fbS2 ( bAutomat:=bAutomat, bManual:=bManual,bStop:=bStop,bReset:=bReset, bEnableMove:=bEnableMoveToS2,bBuffering:=bBuffering,
        bDriveMove:=fbS3.bDrivePrev, bSens1:=bSens1s02D2, bSens2:=bSens1s02D1,bSensFork:= bSens1s01D3, ConvStatusPrev1:=0,
        ConvStatusPrev2:=fbS1.ConvStatus, bButtConv:= bButt1s02, bButtConvRev:=bButt1s02Rev, bButtMove:=bButt1s01_s02,
         bDirect:=bDirect	,bReverse:=bReverse,   ConvStatusNext1:= fbS3.ConvStatus1, ConvStatusNext2:= fbS3.ConvStatus2,
		 bEnableMove3:=bEnableMove3_2(*fbDelayEnableMove3_2.Q*), bEnableMove2:= iCounterPallets>1,  //bSensFreePrev2:=fbS1.bSensFree,
	    bMove1:=bMove1s01_s02_1, bMove2:=bMove2, bMove3:=bMove1s02_1_s02_2, 
        bLongMove1=> bLongMove1s01_s02_1,bLongMove3=> bLongMove1s02_1_s02_2  );

	    bEnableMoveToS3:= NOT bMove1s03_2_s04_1 AND NOT bMove1s03_s04 AND NOT bMove1s01_s02_1 AND NOT bMove1s02_1_s02_2;
 
		
		bEnableMove3_3 := (fbS6.ConvStatus=0 OR fbS5.ConvStatus=0) AND fbS4.ConvStatus1=0 AND fbS4.ConvStatus2=0 
       AND NOT (bMove1s03_2_s04_1 OR bMove1s03_s04 OR bMove1s04_1_s04_2 OR bMove1s05_s06 OR bMove1s04_2_s05);
		  fbDelayEnableMove3_3(IN:=bEnableMove3_3, PT:=T#0.3S);
		  
fbS3 ( bAutomat:=bAutomat, bManual:=bManual,bStop:=bStop,bReset:=bReset, bEnableMove:=bEnableMoveToS3,bBuffering:=bBuffering,
        bDriveMove:=fbS4.bDrivePrev, bSens1:=bSens1s03D2, bSens2:=bSens1s03D1,ConvStatusPrev1:=fbS2.ConvStatus1,
        ConvStatusPrev2:=fbS2.ConvStatus2, bButtConv:= bButt1s03, bButtConvRev:=bButt1s03Rev, bButtMove:=bButt1s02_s03, 
		 bDirect:=bDirect	,bReverse:=bReverse,   ConvStatusNext1:= fbS4.ConvStatus1, ConvStatusNext2:= fbS4.ConvStatus2,
		 bEnableMove3:=fbDelayEnableMove3_3.Q,  bEnableMove2:= TRUE,  //bSensFreePrev1:=fbS2.bSensFree1, bSensFreePrev2:=fbS2.bSensFree2,
	    bMove1:=bMove1s02_2_s03_1, bMove2:=bMove1s02_s03, bMove3:=bMove1s03_1_s03_2, 
        bLongMove1=> bLongMove1s02_2_s03_1,bLongMove2=>bLongMove1s02_s03, bLongMove3=> bLongMove1s03_1_s03_2 );	  
	  
	    bEnableMoveToS4:= NOT bMove1s04_2_s05 AND NOT bMove1s02_2_s03_1 AND NOT bMove1s03_1_s03_2;
 
		
		
		bEnableMove3_4 := fbS6.ConvStatus=0 OR fbS5.ConvStatus=0 AND NOT (bMove1s05_s06 OR bMove1s04_2_s05);
		fbDelayEnableMove3_4(IN:=bEnableMove3_4, PT:=T#0.3S);
		
fbS4 ( bAutomat:=bAutomat, bManual:=bManual,bStop:=bStop,bReset:=bReset, bEnableMove:=bEnableMoveToS4,bBuffering:=bBuffering,
        bDriveMove:=fbS5.bDrivePrev AND bSens1s05D2, bSens1:=bSens1s04D2, bSens2:=bSens1s04D1,ConvStatusPrev1:=fbS3.ConvStatus1,
        ConvStatusPrev2:=fbS3.ConvStatus2, bButtConv:= bButt1s04, bButtConvRev:=bButt1s04Rev, bButtMove:=bButt1s03_s04,
         bDirect:=bDirect	,bReverse:=bReverse,   ConvStatusNext1:= fbS5.ConvStatus,
		 bEnableMove3:=fbDelayEnableMove3_4.Q,  bEnableMove2:= TRUE, // bSensFreePrev1:=fbS3.bSensFree1, bSensFreePrev2:=fbS3.bSensFree2,
	    bMove1:=bMove1s03_2_s04_1, bMove2:=bMove1s03_s04, bMove3:=bMove1s04_1_s04_2, 
         bLongMove1=>bLongMove1s03_2_s04_1,bLongMove2=>bLongMove1s03_s04, bLongMove3=> bLongMove1s04_1_s04_2  );	  
	
  		
		bEnableRead := NOT bMove1s05_s06 AND NOT bMove1s03_2_s04_1 AND NOT bMove1s04_1_s04_2 AND NOT bMove1s03_s04 ;
		
fbLoadScan (bAutomat:=bAutomat,bEnable:=bEnableRead, iConvStatus:=fbS4.ConvStatus2, 
        sInID:=sScanID_1, stLoad:=stLoadS4_1, bReadScan:=bReadScan_1, 
        bRequestID=>bRequestID_1,bEnableReadyID=>bEnableReadyID, bOverflowID=>bOverflow_CTU_ID1,
		bSetVal:=bSetVal_ID1, bResetCTU:=bResetCTU_ID1, bCountNoRead=>bCountNoRead_ID1);		 
		
						
	    bEnableMoveToS5:= NOT bMove1s05_s06 AND NOT bMove1s03_2_s04_1 AND NOT bMove1s04_1_s04_2  AND bEnableReadyID;
	  
fbS5 ( bAutomat:=bAutomat, bManual:=bManual,bStop:=bStop,bReset:=bReset, bEnableMove:= bEnableMoveToS5,
        bDriveMove:=fbS6.bDrivePrev, bSens1:=bSens1s05D2, bSens2:=bSens1s05D1, bStopSecPlace:=TRUE,
        bButtConv:= bButt1s05,bButtConvRev:=bButt1s05Rev, ConvStatusPrev := fbS4.ConvStatus2,
		 bDirect:=bDirect	,bReverse:=bReverse,
		bSensFreePrev:= bSens1s04D1, bMove:=bMove1s04_2_s05,bLongMove=>bLongMove1s04_2_s05, );  
	  	
	
		bEnableWeight := NOT bMove1s04_2_s05 AND NOT bMove1s05_s06 ;
		
fbLoadWeight (bAutomat:=bAutomat,bEnable:=bEnableWeight,bMove:=bMove1s04_2_s05, iConvStatus:=fbS5.ConvStatus, stLoadIn:=stLoadS4_1,
        (*sInWeight:=sWeight_1*)rInWeight:= Massa_1_Gramms   ,  stLoad:=stLoadS5_1, stLoadMove:=stLoadS4_5_1, 
        (*bRequestWeight=>bRequestWeight_1,*) bEnableReadyData=>bEnableReadyData, bOverflowWeight=>bOverflow_CTU_Weight1,
		  bCountNoReadWeight=>bCountNoRead_Weight1, bSetValWeight:=bSetVal_Weight1, bResetCTUWeight:=bResetCTU_Weight1);	
		
			
	    bEnableMoveToS6:= NOT bMove1s04_2_s05   AND bEnableReadyData ;
	  
fbS6 ( bAutomat:=bAutomat, bManual:=bManual,bStop:=bStop,bReset:=bReset, bEnableMove:= bEnableMoveToS6,
        bSens1:=TRUE, bSens2:=bSens1s06D1, (*bSensFork:= bSens1s06D2, *)bButtConv:= bButt1s06, bButtConvRev:=bButt1s06Rev,
		 bDirect:=bDirect	,bReverse:=bReverse,bLastPlace:=TRUE,bLongMove=>bLongMove1s05_1s06,
	    bMove:=bMove1s05_s06,ConvStatusPrev := fbS5.ConvStatus,bSensFreePrev := bSensFreePrevS6);  
		
		bSensFreePrevS6 := fbS6.ConvStatus = 0;
		
		
fbLoadDataToWMS(bAutomat:=bAutomat,stLoadIn:=stLoadS5_1, bEnable:=NOT bMove1s05_s06, 
iConvStatus:=fbS6.ConvStatus, bMove	:=bMove1s05_s06, stLoadMove:=  stLoadS5_6_1, stLoad:=stLoadS6_1,
sMessageOut=>sMessageOut1, bMessageReady:=bMessageReady1	);		
		
		
	  
bDrive1s01M1    := fbS1.bDrive 		AND bDirect ;
bDrive1s01M1Rev := fbS1.bDriveRev 		AND bReverse AND bSens1s01D2;
bDrive1s02M1    := fbS2.bDrive 		AND bDirect ;
bDrive1s02M1Rev := fbS2.bDriveReverse 	AND bReverse;
bDrive1s03M1    := fbS3.bDrive 		AND bDirect ;
bDrive1s03M1Rev := fbS3.bDriveReverse 	AND bReverse;
bDrive1s04M1    := fbS4.bDrive 		AND bDirect ;
bDrive1s04M1Rev := fbS4.bDriveReverse 	AND bReverse;  
bDrive1s05M1    := fbS5.bDrive 		AND bDirect ;
bDrive1s05M1Rev := fbS5.bDriveRev 		AND bReverse;
bDrive1s06M1    := fbS6.bDrive 		AND bDirect AND bSens1s06D1;
bDrive1s06M1Rev := fbS6.bDriveRev 		AND bReverse;

END_PROGRAM

// ---- POUs/FB/FBconv/FB_ConvPlace.TcPOU
FUNCTION_BLOCK FB_ConvPlace
VAR_INPUT
	bFirstPlace:BOOL:=FALSE;
	bLastPlace:BOOL:=FALSE;
	bAutomat: BOOL;
	bStopSecPlace: BOOL;
	bEnableMove: BOOL;
	ConvStatusPrev: BYTE;
	bManual: BOOL;
	bDriveMove: BOOL;
	bSens1: BOOL;
	bSens2: BOOL;
	bSens3: BOOL := TRUE;
	bSensFork: BOOL := FALSE;
	tBusy: TIME := TIME#10ms;
	tFree: TIME := TIME#2s800ms;
	tLongMove: TIME := TIME#15s0ms;
	bReset: BOOL := FALSE;
	bStop: BOOL;
	bSensFreePrev: BOOL;
	bSensFreeNext: BOOL;
	bButtConv: BOOL;
	bButtConvRev: BOOL;
	bButtMove: BOOL;
	 bDirect: BOOL;
	bReverse: BOOL;
END_VAR
VAR_OUTPUT
	bDrive: BOOL;
	bDriveRev: BOOL;
	ConvStatus: BYTE;
	bDrivePrev: BOOL;
	bLongMove: BOOL;
	bSensFree: BOOL;
	bReqMove: BOOL;
	bForkFree: BOOL;
END_VAR
VAR
	fbBusy1: FB_Busy1;
	fbBusy2: FB_Busy1;
	fbBusy3: FB_Busy1;
	fbBusyFork: FB_Busy2;
	fbButt: FB_ButtonToggle;
	fbButtRev: FB_ButtonToggle;
	bDriveManu: BOOL;
	bResManu: BOOL;
	bDriveManuRev: BOOL;
	fbLongMove: TON;
	bDriveConv: BOOL;
	fbButtMove: R_TRIG;
	bDriveConvRev: BOOL;
END_VAR
VAR_IN_OUT
	bMove: BOOL;
END_VAR






     (* определение заполненности конвейерного места*)
    fbBusy1 ( bSens:= bSens1,  tFree:=  tFree ,   tBusy:= tBusy , Reset := bReset ) ;
	fbBusy2 ( bSens:= bSens2,  tFree:=   tFree ,   tBusy:=  tBusy , Reset := bReset ) ;
	fbBusy3 ( bSens:= bSens3,  tFree:=   tFree ,   tBusy:=  tBusy , Reset := bReset ) ;
	fbBusyFork( bSens:= bSensFork,  tFree:=   T#10s ,   tBusy:= T#0s , Reset := bReset ) ;
	IF  NOT fbBusy1.ConvBusy AND NOT  fbBusy2.ConvBusy AND NOT  fbBusy3.ConvBusy THEN ConvStatus := 0;
	ELSIF fbBusy1.ConvBusy AND NOT  fbBusy2.ConvBusy THEN ConvStatus := 1;
	ELSIF NOT  fbBusy1.ConvBusy AND   fbBusy2.ConvBusy THEN ConvStatus := 2;
	ELSIF fbBusy1.ConvBusy AND   fbBusy2.ConvBusy THEN ConvStatus := 3;
	END_IF
	
	bForkFree:= NOT fbBusyFork.ConvBusy;
	
	bSensFree:= bSens1 AND bSens2 AND bSens3;
	
	(* включение двигателя*)
     bDrive:= NOT bStop AND (  bDriveMove OR bDriveConv  OR  bDriveManu );
	  bDriveRev:= NOT bStop AND bDriveManuRev;
	
    (* включение двигателя в ручном режиме *)
	bResManu := bReset OR NOT bManual ;
	fbButt (bButt := bButtConv , bEnable := bManual AND NOT bDriveManuRev AND bDirect , bReset := bResManu OR NOT bDirect
OR bDirect AND bLastPlace AND NOT bSens2)  ;
     bDriveManu := fbButt.bOutB;
	fbButtRev (bButt := bButtConvRev  , bEnable :=  bManual  AND NOT bDriveManu AND bReverse, bReset := bResManu OR NOT bReverse
OR bReverse AND bFirstPlace AND NOT bSens1)  ;
 bDriveManuRev := fbButtRev.bOutB;

	(* включение перемещения*)

bReqMove:= bAutomat  AND  (ConvStatusPrev = 2  OR ConvStatusPrev =3) AND ConvStatus =0 AND  NOT fbBusyFork.ConvBusy ;

	IF    bEnableMove   AND  bReqMove
	 THEN  bMove := TRUE ;
	END_IF
	
	(* включение двигателей при перемещении *)
	bDriveConv:=   NOT bStop AND bMove  AND NOT  (ConvStatus = 2 OR ConvStatus = 3)  ;
	bDrivePrev := NOT bStop AND bMove AND NOT  (ConvStatus = 2 OR ConvStatus = 3) AND NOT (ConvStatusPrev = 0) ;
	

	
	
	(* выключение перемещения*)
	IF   bMove  AND ((*ConvStatusPrev = 0*) bSensFreePrev  OR bStopSecPlace ) AND  (ConvStatus = 2 OR ConvStatus = 3)  THEN bMove := FALSE ;
	END_IF
	
	(* долгое перемещение*)
	fbLongMove(IN := NOT bStop AND bMove , PT := tLongMove);
	 bLongMove:= fbLongMove.Q;
	 
	 (* включение-выключение перемещения кнопкой*)
	 
	fbButtMove (CLK :=bButtMove (*AND bManual*));
	IF fbButtMove.Q AND bManual THEN IF   NOT bMove  THEN bMove := TRUE;
         ELSIF bMove THEN  
      bMove := FALSE;
	END_IF
    END_IF
		
		


	 
		
		
	 IF bReset THEN 
     bMove := FALSE ; 
	  END_IF

END_FUNCTION_BLOCK

// ---- POUs/FB/FBauxiliary/FB_Busy1.TcPOU
FUNCTION_BLOCK FB_Busy1
VAR_INPUT
	bSens	 :BOOL;
	tBusy	 :TIME;
	tFree	 :TIME;
	Reset	 :BOOL;
END_VAR
VAR_OUTPUT
	ConvBusy :BOOL := TRUE;
END_VAR
VAR
	Timer1	 :TON;
	Timer2	 :TON;
END_VAR

Timer1 (IN := NOT bSens, PT := tBusy);
IF Timer1.Q THEN ConvBusy := TRUE;
END_IF
Timer2 (IN :=     bSens, PT := tFree);
IF Timer2.Q (*OR Reset*) THEN ConvBusy := FALSE;
END_IF

END_FUNCTION_BLOCK

// ---- POUs/FB/FBauxiliary/FB_Busy2.TcPOU
FUNCTION_BLOCK FB_Busy2
VAR_INPUT
	bSens	 :BOOL;
	tBusy	 :TIME;
	tFree	 :TIME;
	Reset	 :BOOL;
END_VAR
VAR_OUTPUT
	ConvBusy :BOOL;
END_VAR
VAR
	Timer1	 :TON;
	Timer2	 :TON;
END_VAR

Timer1 (IN := 	  bSens, PT := tBusy);
IF Timer1.Q THEN ConvBusy := TRUE;
END_IF
Timer2 (IN := NOT bSens, PT := tFree);
IF Timer2.Q (*OR Reset*) THEN ConvBusy := FALSE;
END_IF

END_FUNCTION_BLOCK

// ---- POUs/FB/FBconv/FB_ConvPlaceDouble.TcPOU
FUNCTION_BLOCK FB_ConvPlaceDouble
VAR_INPUT
	bStopSecPlace: BOOL;
	bStartAutomat: BOOL;
	bAutomat: BOOL;
	bManual: BOOL;
	bReset: BOOL := FALSE;
	bStop: BOOL;
	bEnableMove: BOOL;
	ConvStatusPrev1: BYTE;
	ConvStatusPrev2: BYTE;
	bDriveMove: BOOL;
	bButtConv: BOOL;
	bButtConvRev: BOOL;
	bButtMove: BOOL;
	bSens1: BOOL;
	bSens2: BOOL;
	bSens3: BOOL := TRUE;
	bSensFork: BOOL := FALSE;
	tBusy: TIME := TIME#10ms;
	tFree: TIME := TIME#2s800ms;
	tLongMove: TIME := TIME#30s0ms;
	bBuffering: BOOL;
	 bDirect: BOOL;
	bReverse: BOOL;
	ConvStatusNext1: BYTE;
	ConvStatusNext2: BYTE;
	bEnableMove3:BOOL;
	bEnableMove2:BOOL;
	
	bSensFreePrev1:BOOL;
	bSensFreePrev2:BOOL;
END_VAR
VAR_OUTPUT
	bDrive: BOOL;
	bDriveReverse: BOOL;
	ConvStatus2: BYTE;
	ConvStatus1: BYTE;
	bDrivePrev: BOOL;
	bLongMove1: BOOL;
	bLongMove2: BOOL;
	bLongMove3: BOOL;
	bSensFree1:BOOL;
	bSensFree2:BOOL;
END_VAR
VAR
	fbBusy1: FB_Busy1;
	fbBusy2: FB_Busy1;
	fbBusyFork: FB_Busy2;
	fbButt: FB_ButtonToggle;
	fbButtReverse: FB_ButtonToggle;
	bDriveManu: BOOL;
	bResManu: BOOL;
	bDriveManuReverse: BOOL;
	bDriveConv1: BOOL;
	bDriveConv2: BOOL;
	bDriveConv3: BOOL;
	bDriveConv: BOOL;
	bDrivePrev1: BOOL;
	bDrivePrev2: BOOL;
	fbLongMove1: TON;
	fbLongMove2: TON;
	fbLongMove3: TON;
	fbButtMove: R_TRIG;
	fbStartAutomat: R_TRIG;
	bStartConv: BOOL;
	fbConvBusy1Puls: R_TRIG;
	fbConvBusy2Puls: R_TRIG;
	fbStartTimer: TON;
	fbFinStartAutomat: F_TRIG;
	bPermMove1: BOOL;
	bPermMove2: BOOL;
	bPermMove3: BOOL;

END_VAR
VAR_IN_OUT
	bMove1: BOOL;
	bMove2: BOOL;
	bMove3: BOOL;
END_VAR

fbBusy1 ( bSens := bSens1, tFree := tFree, tBusy := tBusy, Reset := bReset);
fbBusy2 ( bSens := bSens2, tFree := tFree, tBusy := tBusy, Reset := bReset);
fbBusyFork( bSens:= bSensFork,  tFree:=   T#10S ,   tBusy:= T#0S , Reset := bReset ) ;

 bSensFree1:= bSens1;    
 bSensFree2:= bSens2; 

IF NOT fbBusy1.ConvBusy THEN ConvStatus1 := 0;
	ELSE
		ConvStatus1 := 2;
END_IF

IF NOT fbBusy2.ConvBusy  THEN ConvStatus2 := 0;
	ELSE
		ConvStatus2 := 2;
END_IF

bDrive := NOT bStop AND (bDriveMove OR bDriveConv OR bDriveManu OR bStartConv);
bDriveReverse := NOT bStop AND bDriveManuReverse;

bResManu := bReset OR NOT bManual;
fbButt (bButt := bButtConv AND bManual AND NOT bDriveManuReverse AND bDirect, bReset := bResManu  OR NOT bDirect); 
bDriveManu := fbButt.bOutB;
fbButtReverse (bButt := bButtConvRev AND bManual AND NOT bDriveManu AND bReverse, bReset := bResManu  OR NOT bReverse);
 bDriveManuReverse := fbButtReverse.bOutB;

(* Перемещения*)
(* Условия включения перемещения*)
bPermMove1:= ConvStatusPrev1=0 AND ConvStatus2=0  AND NOT bMove2  AND NOT bMove3;

IF  bAutomat AND bEnableMove AND bPermMove1 AND (ConvStatusPrev2 = 2 OR ConvStatusPrev2 = 3) AND ConvStatus1 = 0 AND  NOT fbBusyFork.ConvBusy
	THEN  bMove1 := TRUE;
END_IF

(* Выключение перемещения bMove1*)
IF  bMove1 AND (ConvStatusPrev2 = 0 OR bStopSecPlace (*OR bSensFreePrev2*)) AND (ConvStatus1 = 2 OR ConvStatus1 = 3) THEN bMove1 := FALSE;
END_IF





bPermMove2 := (( ConvStatusPrev1=2 OR ConvStatusPrev1=3) AND ConvStatus1=0 OR  ConvStatusPrev1=0 AND  (ConvStatus1 = 2 OR
ConvStatus1 = 3)) AND NOT bMove1  AND NOT bMove3 AND bEnableMove2;

IF  bAutomat AND bEnableMove AND bPermMove2 AND (ConvStatusPrev2 = 2 OR ConvStatusPrev2 = 3) AND ConvStatus2 = 0 
	THEN  bMove2 := TRUE;
END_IF


(* Выключение перемещения bMove2*)
IF  bMove2 AND (ConvStatusPrev2 = 0 OR bStopSecPlace (*OR bSensFreePrev2*)) AND (ConvStatus2 = 2 OR ConvStatus2 = 3) THEN bMove2 := FALSE;
END_IF

//bPermMove3 := (ConvStatusNext1=0 AND ConvStatusNext2=0  OR (ConvStatusNext1=2 OR ConvStatusNext1=3) AND ConvStatusNext2=0 )
//AND NOT bMove1 AND NOT bMove2;
bPermMove3 := (NOT (( ConvStatusPrev2=2 OR ConvStatusPrev2=3) AND ConvStatusPrev1=0) AND NOT bBuffering OR
bBuffering AND 	bEnableMove3)  AND NOT bMove1 AND NOT bMove2;

IF  bAutomat AND bEnableMove AND bPermMove3 AND (ConvStatus1 = 2 OR ConvStatus1 = 3) AND ConvStatus2 = 0 
	THEN bMove3 := TRUE;
END_IF

(* Выключение перемещения bMove3*)
IF  bMove3 AND (ConvStatus1 = 0 OR bStopSecPlace (*OR bSens1*)) AND (ConvStatus2 = 2 OR ConvStatus2 = 3) THEN bMove3 := FALSE;
END_IF




(* Включение двигателей *)
bDriveConv1 := NOT bStop AND bMove1 AND NOT (ConvStatus1 = 2 OR ConvStatus1 = 3);
bDriveConv2 := NOT bStop AND bMove2 AND NOT (ConvStatus2 = 2 OR ConvStatus2 = 3);
bDriveConv3 := NOT bStop AND bMove3 AND NOT (ConvStatus2 = 2 OR ConvStatus2 = 3);
	
bDriveConv := bDriveConv1 OR bDriveConv2 OR bDriveConv3;

bDrivePrev1 := NOT bStop AND bMove1 AND NOT (ConvStatus1 = 2 OR ConvStatus1 = 3) AND NOT (ConvStatusPrev2 = 0);
bDrivePrev2 := NOT bStop AND bMove2 AND NOT (ConvStatus2 = 2 OR ConvStatus2 = 3) AND NOT ((ConvStatusPrev1 = 0)AND(ConvStatusPrev2 = 0)) ;
	
bDrivePrev := bDrivePrev1 OR bDrivePrev2 ;

(* Долгое перемещение*)
fbLongMove1(IN := NOT bStop AND bMove1, PT := tLongMove);
bLongMove1 := fbLongMove1.Q;
fbLongMove2(IN := NOT bStop AND bMove2, PT := tLongMove);
bLongMove2 := fbLongMove2.Q;
fbLongMove3(IN := NOT bStop AND bMove3, PT := tLongMove);
bLongMove3 := fbLongMove3.Q;

(* Включение-выключение перемещения кнопкой*)
fbButtMove (CLK :=bButtMove (*AND bManual*));
IF fbButtMove.Q THEN 
	IF NOT bMove2 AND bManual THEN bMove2 := TRUE;
		ELSIF bMove2 THEN  
      bMove2 := FALSE;
	END_IF
   // bButtMove := FALSE;
END_IF

IF  bReset THEN bMove1 := FALSE; bMove2 := FALSE; bMove3 := FALSE; bStartConv := FALSE; 
	
END_IF

(*
(* Начальный режим*)
	fbStartAutomat (CLK := bStartAutomat);
IF 	fbStartAutomat.Q THEN 
IF NOT bReverse 
THEN 
IF (ConvStatus1=2 OR ConvStatus1=3)AND ConvStatusNext =1          THEN
	bStartConvReverse := TRUE;
END_IF

ELSE  bStartConvReverse := TRUE;
(* IF  NOT (ConvStatus1=2 OR ConvStatus1=3)AND ConvStatusNext =1 
THEN  bStartConvReverse := TRUE;
END_IF*)
END_IF
END_IF

	fbConvBusy1Puls (CLK := fbBusy1.ConvBusy);
//	fbConvBusy2Puls (CLK := fbBusy2.ConvBusy);

//	fbStartTimer (IN := bStartConv, PT := tStartTimer);
	fbStartTimerReverse (IN := bStartConvReverse, PT := tStartTimer);

(*IF    (bFinalConv  AND (ConvStatus = 3 OR ConvStatus = 2) OR NOT bFinalConv AND ((ConvStatus = 3 OR ConvStatus = 2) AND (ConvStatusNext = 3 OR ConvStatusNext = 2)) OR fbConvBusy2Puls.Q OR fbStartTimer.Q)
OR NOT bStartAutomat THEN  bStartConv := FALSE;
END_IF*)

IF 	  (bStartConvReverse AND (bFinalConvReverse AND (ConvStatus = 3 OR ConvStatus = 1) OR NOT bFinalConvReverse AND ((ConvStatus = 3 OR ConvStatus = 1) AND (ConvStatusPrev = 3 OR ConvStatusPrev = 1)) OR fbConvBusy1Puls.Q OR fbStartTimerReverse.Q))
OR NOT bStartAutomat THEN bStartConvReverse := FALSE;
END_IF

fbFinStartAutomat(CLK:=bStartAutomat);
IF fbFinStartAutomat.Q AND (ConvStatus1=2 OR ConvStatus1=3)AND ConvStatusNext =1   THEN
	bMoveReverse:=TRUE;
END_IF
*)

END_FUNCTION_BLOCK

// ---- POUs/ProcessingLoadData/FB_LoadScan.TcPOU
FUNCTION_BLOCK FB_LoadScan
VAR_INPUT
	bEnable			:BOOL;
	iConvStatus		:BYTE;
	bAutomat		:BOOL;
	
	bResetCTU		:BOOL;		
	bSetVal			:WORD;			
END_VAR
VAR_OUTPUT
	bEnableReadyID	:BOOL;
	bRequestID		:BOOL;
	bCountNoRead	:WORD;		//Кол-во несчитываний
	bOverflowID		:BOOL;		//Переполнение счетчика несчитываний ID
END_VAR
VAR
	fbPulsRequest	:R_TRIG;
	bStartRequest	:BOOL;
	fbDelayRead		:TON;
	WaitingID		:TON;
	bNoRead			:BOOL;		//Несчитывание
	bWriteIDgood	:BOOL;
	fbPulsNoread 	:R_TRIG;
	CTU 			:CTU;		//Счетчик
END_VAR
VAR_IN_OUT	
	stLoad			:ST_LoadData;
	bReadScan		:BOOL;
	sInID			:STRING;
END_VAR


bStartRequest:= bEnable AND bAutomat AND (iConvStatus=2 OR iConvStatus=3);

bEnableReadyID 	R= NOT bStartRequest;
bRequestID 	   	R= NOT bStartRequest  OR bReadScan;
bNoRead 		R= NOT bStartRequest;
bWriteIDgood    R= NOT bStartRequest;

fbPulsRequest(CLK:=bStartRequest);
IF fbPulsRequest.Q THEN
	bRequestID:=TRUE;
	bReadScan:=FALSE;
END_IF

fbDelayRead(IN:=bReadScan, PT:=T#0.3S);

WaitingID(IN:= bRequestID , PT:=T#3S);
bNoRead S= WaitingID.Q ;

fbPulsNoread(CLK:=bNoRead);

CTU(CU:=fbPulsNoread.Q, RESET:=bResetCTU, PV:=bSetVal);
bCountNoRead:=CTU.CV;

IF bReadScan AND NOT (bCountNoRead>=bSetVal) THEN
	stLoad.sID:= sInID;
	
	IF stLoad.sID<>'' OR fbDelayRead.Q THEN	
		bWriteIDgood:=TRUE;
		bReadScan:=FALSE;
	END_IF	
END_IF
bEnableReadyID S= bWriteIDgood OR bNoRead;

IF iConvStatus=0 THEN
	stLoad.sID:= '';
	stLoad.sWeight:= '';
	sInID:='';
END_IF

(*IF bCountNoRead>=bSetVal THEN bOverflowID:=TRUE;
	ELSE bOverflowID:=FALSE;
END_IF*)

END_FUNCTION_BLOCK

// ---- POUs/ProcessingLoadData/FB_LoadWeight.TcPOU
FUNCTION_BLOCK FB_LoadWeight
VAR_INPUT
	stLoadIn			:ST_LoadData;
	bEnable				:BOOL;
	iConvStatus			:BYTE;
	bAutomat			:BOOL;
	
	rInWeight			:DINT;;
	bMove				:BOOL;
	bReadWeight     	:BOOL;
	
	bResetCTUWeight		:BOOL;	//Очистка счетчика невзвешиваний	
	bSetValWeight		:WORD;	//Заданное значение разрешенных ошибок
END_VAR
VAR_OUTPUT
	bEnableReadyData	:BOOL;
	bRequestWeight		:BOOL;
	bCountNoReadWeight	:WORD;		//Кол-во несчитываний
	bOverflowWeight		:BOOL;		//Переполнение счетчика несчитываний весов
END_VAR
VAR
	fbPulsRequest		:R_TRIG;
	bStartRequest		:BOOL;
	fbPulsReadWeight	:R_TRIG;
	fbDelayWeight		:TON;
	fbStartMove			:R_TRIG;
	fbFinMove			:F_TRIG;
	bReadySt			:BOOL;
	bStartMove			:BOOL;
	bEndMove			:BOOL;
	sInWeight			:STRING;
	
	WaitingWeight		:TON;
	bNoReadWeight		:BOOL;		//Несчитывание
	bWriteWeightGood	:BOOL;
	fbPulsNoreadWeight 	:R_TRIG;
	CTU 				:CTU;		//Счетчик
END_VAR

VAR_IN_OUT
	stLoadMove      	:ST_LoadData;
	stLoad				:ST_LoadData;
//	bReadWeight			:BOOL;
END_VAR

fbStartMove(CLK:=bMove);
bStartMove S=fbStartMove.Q;
IF bStartMove THEN 
	stLoadMove := stLoadIn;
	IF stLoadMove.sID=stLoadIn.sID  AND stLoadMove.sWeight=stLoadIn.sWeight  THEN
		bStartMove:=FALSE;
	END_IF
END_IF

fbFinMove(CLK:=bMove);
bEndMove S= fbFinMove.Q;
IF bEndMove THEN 
	stLoad := stLoadMove;
	IF stLoadMove.sID=stLoad.sID  AND stLoadMove.sWeight=stLoad.sWeight  THEN
		bEndMove:=FALSE;
	END_IF
END_IF
//bReadySt := stLoad.sID = stLoadIn.sID  AND stLoad.sWeight = stLoadIn.sWeight;

bStartRequest:= bEnable AND bAutomat AND (iConvStatus=2 OR iConvStatus=3) AND NOT bEndMove;

bEnableReadyData 	R= NOT bStartRequest;
bRequestWeight 		R= NOT bStartRequest;
bNoReadWeight		R= NOT bStartRequest;

fbPulsRequest(CLK:=bStartRequest);
IF fbPulsRequest.Q THEN
	bRequestWeight:=TRUE;
END_IF

WaitingWeight(IN:= bRequestWeight, PT:=T#2S);
bNoReadWeight S= WaitingWeight.Q ;

fbPulsNoreadWeight(CLK:=bNoReadWeight);

CTU(CU:=fbPulsNoreadWeight.Q, RESET:=bResetCTUWeight, PV:=bSetValWeight);
bCountNoReadWeight:=CTU.CV;

fbDelayWeight(IN:=bRequestWeight(*bReadWeight*), PT:=T#0.3S);

sInWeight:= DINT_TO_STRING(rInWeight);
IF bRequestWeight(*bReadWeight  AND bReadySt*)AND NOT (bCountNoReadWeight=bSetValWeight) THEN
	stLoad.sWeight:= sInWeight;
	
	IF stLoad.sWeight<>'' OR fbDelayWeight.Q THEN	
		bWriteWeightGood	:=TRUE;	
		bRequestWeight		:=FALSE;
	END_IF	
END_IF

bEnableReadyData S= bWriteWeightGood OR bNoReadWeight;

IF iConvStatus=0 THEN
	stLoad.sID:= '';
	stLoad.sWeight:= '';
END_IF

IF bCountNoReadWeight>=bSetValWeight THEN bOverflowWeight:=TRUE;
	ELSE bOverflowWeight:=FALSE;
END_IF

END_FUNCTION_BLOCK

// ---- POUs/ExchangeWMS/FB_LoadDataToWMS.TcPOU
FUNCTION_BLOCK FB_LoadDataToWMS
VAR_INPUT
	stLoadIn		:ST_LoadData;
	bEnable			:BOOL;
	iConvStatus		:BYTE;
	bAutomat		:BOOL;
	bMove			:BOOL;
	
END_VAR
VAR_OUTPUT
	sMessageOut:T_MaxString;
	
END_VAR
VAR
	fbStartMove		:R_TRIG;
	fbFinMove		:F_TRIG;
	
	bStartMove:BOOL;
	bEndMove:BOOL;
	fbDelayStartMove:TON;
	fbDelayFinMove:TON;
	bReadySend: BOOL;
	
	fbCreateMessage: FB_CreateMessage;
END_VAR
VAR_IN_OUT
	stLoadMove      :ST_LoadData;
	stLoad			:ST_LoadData;
     bMessageReady:BOOL;
END_VAR

fbStartMove(CLK:=bMove);
bStartMove S=fbStartMove.Q;
fbDelayStartMove(IN:=bStartMove,PT:=T#0.3S);
IF bStartMove THEN 
	stLoadMove := stLoadIn;
	IF stLoadMove.sID=stLoadIn.sID  AND  stLoadMove.sWeight=stLoadIn.sWeight OR fbDelayStartMove.Q  THEN
		bStartMove:= FALSE;
	END_IF
END_IF


fbFinMove(CLK:=bMove);
bEndMove S= fbFinMove.Q;
fbDelayFinMove(IN:=bEndMove,PT:=T#0.3S);
IF bEndMove THEN 
	stLoad := stLoadMove;
	IF stLoadMove.sID=stLoad.sID   AND  stLoadMove.sWeight=stLoad.sWeight  OR fbDelayFinMove.Q  THEN
		bEndMove:= FALSE;
	END_IF
END_IF


bReadySend:=bAutomat AND (iConvStatus=2 OR iConvStatus=3) AND NOT bEndMove;

fbCreateMessage(stLoad:=stLoad, bCreateMessage:=bReadySend, sMessageOut=>sMessageOut,
bMessageReady:= bMessageReady );

END_FUNCTION_BLOCK

// ---- POUs/ExchangeWMS/FB_CreateMessage.TcPOU
FUNCTION_BLOCK FB_CreateMessage
VAR_INPUT
	stLoad		:ST_LoadData;
	bCreateMessage :BOOL;
END_VAR
VAR_OUTPUT
	sMessageOut:T_MaxString;
	
END_VAR
VAR
sTemplateMessage:T_MaxString:='|MsgNam=WMS.TEGEW|TrxId=|RFIDNAM=|DzTrn=|ArtGewBru=|';
fbPulsCreateMessage:R_TRIG;
sTrxId:STRING;
i :INT;
sMessage :T_MaxString;
iPosRFID:INT;
iPosTime:INT;
iPosBrutto:INT;
	

fbFileOpen:FB_FileOpen;
END_VAR
VAR PERSISTENT
iCountTrxId: UINT;
END_VAR
VAR_IN_OUT
	bMessageReady:BOOL;
END_VAR






fbPulsCreateMessage(CLK:=bCreateMessage);

IF fbPulsCreateMessage.Q THEN
	iCountTrxId:= iCountTrxId+1;
	i:=1;
END_IF
CASE i OF
	0:  ;
	
	1:
bMessageReady:=FALSE;	
sTrxId:= INT_TO_STRING(iCountTrxId);	

sMessage:= INSERT(sTemplateMessage,	sTrxId,24);
iPosRFID:= FIND(sMessage,'RFIDNAM=');
sMessage:= INSERT(sMessage,	stLoad.sID,iPosRFID+7);
iPosTime:= FIND(sMessage,'DzTrn=');
sMessage:= INSERT(sMessage,	sSystemTime,iPosTime+5);
iPosBrutto:= FIND(sMessage,'ArtGewBru=');
sMessage:= INSERT(sMessage,	stLoad.sWeight,iPosBrutto+9);

	i:=3;
	
	3:
sMessageOut:=	sMessage;
IF 	sMessageOut=sMessage THEN
	bMessageReady:=TRUE;
	i:=0;
END_IF

	
END_CASE

END_FUNCTION_BLOCK

// ---- POUs/ConvLine2.TcPOU
PROGRAM ConvLine2
VAR_INPUT
	bAutomat		:BOOL;
	bManual			:BOOL;
	bStop			:BOOL;
	bReset			:BOOL := FALSE;
	bDirect			:BOOL;
	bReverse		:BOOL;
	bBuffering		:BOOL;
END_VAR
VAR
	fbS1			:FB_ConvPlace;
	fbS2			:FB_ConvPlaceDouble;
	fbS3			:FB_ConvPlaceDouble;
	fbS4			:FB_ConvPlaceDouble;
	fbS5			:FB_ConvPlace;
	fbS6			:FB_ConvPlace;
	bMove1			:BOOL;
	bMove2			:BOOL;
	bDriveMoveS1	:BOOL;
	bDriveMoveS2	:BOOL;
	bEnableMoveToS1	:BOOL :=TRUE;
	bEnableMoveToS2	:BOOL;
	bEnableMoveToS3	:BOOL;
	bEnableMoveToS4	:BOOL;
	bEnableMoveToS5	:BOOL;
	bEnableMoveToS6	:BOOL;
	bEnableRead		:BOOL;
	bEnableWeight	:BOOL;
	fbLoadScan		:FB_LoadScan;
	fbLoadWeight	:FB_LoadWeight;
	bEnableReadyID	:BOOL;
	bEnableReadyData:BOOL;
	ConvStatusPrev 	:BYTE;
	bSensFreePrevS1 :BOOL;
	bSensFreePrevS5 :BOOL;
	bSensFreePrevS6 :BOOL;
	
	bCountNoRead_ID2		:WORD;		//Кол-во несчитываний RFID
	bSetVal_ID2				:WORD :=10;	//Заданное значение счетчика (максимально допустимое для несчитываний)
	bResetCTU_ID2			:BOOL;		//Сброс счетчика несчитываний
	
	bCountNoRead_Weight2	:WORD;		//Кол-во несчитываний RFID
	bSetVal_Weight2			:WORD :=10;	//Заданное значение счетчика (максимально допустимое для несчитываний)
	bResetCTU_Weight2		:BOOL;		//Сброс счетчика несчитываний
	
	fbLoadDataToWMS: FB_LoadDataToWMS;
	
	
	bEnableMove3_2:BOOL;
	bEnableMove3_3:BOOL;
	bEnableMove3_4:BOOL;
	
	fbFallMove1:R_TRIG;
	bLineFree:BOOL;
	fbFreeS6:R_TRIG;
	
END_VAR
VAR PERSISTENT
	iCounterPallets:INT;
END_VAR







fbS1 ( bAutomat:=bAutomat, bManual:=bManual,bStop:=bStop,bReset:=bReset,tBusy:=T#6S, bDirect:=bDirect	,bReverse:=bReverse,
       	bDriveMove:=fbS2.bDrivePrev, bSens1:=bSens2s01D2, bSens2:=bSens2s01D1, bFirstPlace:=TRUE,
       	bSensFork:= bSens2s01D3, bButtConv:= bButt2s01,bButtConvRev:=bButt2s01Rev,
	  	bMove:=bMove1,ConvStatusPrev:=ConvStatusPrev, bEnableMove := bEnableMoveToS1, bSensFreePrev := bSensFreePrevS1);
		bSensFreePrevS1 := fbS1.ConvStatus = 0;
		
	  	bEnableMoveToS2:= NOT bMove2s02_2_s03_1 AND NOT bMove2s02_s03;
	  
		bLineFree:= fbS3.ConvStatus1=0 AND fbS3.ConvStatus2=0 AND 
      fbS4.ConvStatus1=0 AND fbS4.ConvStatus2=0 AND NOT (bMove2s02_2_s03_1 OR bMove2s02_s03 OR bMove2s03_1_s03_2
      OR bMove2s03_2_s04_1 OR bMove2s03_s04 OR bMove2s04_1_s04_2  OR bMove2s05_s06 OR bMove2s04_2_s05);	 

		
		
	 IF bLineFree AND fbS6.ConvStatus=0 AND fbS5.ConvStatus=0 THEN
	 iCounterPallets:=0;
 END_IF
	  
		fbFallMove1(CLK:=bMove2s02_2_s03_1 OR bMove2s02_s03 )  ;
IF fbFallMove1.Q THEN
	IF bMove2s02_2_s03_1 THEN
iCounterPallets:=iCounterPallets +1;
ELSIF  bMove2s02_s03 THEN 	
	iCounterPallets:=iCounterPallets +2;
END_IF	
END_IF
		fbFreeS6(CLK:=fbS6.ConvStatus=0);
IF fbFreeS6.Q AND iCounterPallets>0 THEN
iCounterPallets:=iCounterPallets -1;	
END_IF

		
		bEnableMove3_2 := (*(fbS6.ConvStatus=0 OR fbS5.ConvStatus=0) AND bLineFree OR *)iCounterPallets<2;
	//  fbDelayEnableMove3_2(IN:=bEnableMove3_2, PT:=T#0.3S);
			
		
		
		
fbS2 ( bAutomat:=bAutomat, bManual:=bManual,bStop:=bStop,bReset:=bReset, bEnableMove:=bEnableMoveToS2,bBuffering:=bBuffering,
        bDriveMove:=fbS3.bDrivePrev, bSens1:=bSens2s02D2, bSens2:=bSens2s02D1,bSensFork:= bSens2s01D3,ConvStatusPrev1:=0,
        ConvStatusPrev2:=fbS1.ConvStatus, bButtConv:= bButt2s02, bButtConvRev:=bButt2s02Rev, bButtMove:=bButt2s01_s02,
        bDirect:=bDirect	,bReverse:=bReverse,
		ConvStatusNext1:= fbS3.ConvStatus1, ConvStatusNext2:= fbS3.ConvStatus2,
	    bMove1:=bMove2s01_s02_1, bMove2:=bMove2s01_s02, bMove3:=bMove2s02_1_s02_2, 
        bEnableMove3:=bEnableMove3_2, bEnableMove2:= iCounterPallets>1, 
        bLongMove1=> bLongMove2s01_s02_1,bLongMove3=> bLongMove2s02_1_s02_2 );

	    bEnableMoveToS3:= NOT bMove2s03_2_s04_1 AND NOT bMove2s03_s04 AND NOT bMove2s01_s02_1 AND NOT bMove2s02_1_s02_2;
 
		
			bEnableMove3_3 := (fbS6.ConvStatus=0 OR fbS5.ConvStatus=0) AND fbS4.ConvStatus1=0 AND fbS4.ConvStatus2=0 
       AND NOT (bMove2s03_2_s04_1 OR bMove2s03_s04 OR bMove2s04_1_s04_2 OR bMove2s05_s06 OR bMove2s04_2_s05);
		
		
		
fbS3 ( bAutomat:=bAutomat, bManual:=bManual,bStop:=bStop,bReset:=bReset, bEnableMove:=bEnableMoveToS3,bBuffering:=bBuffering,
        bDriveMove:=fbS4.bDrivePrev, bSens1:=bSens2s03D2, bSens2:=bSens2s03D1,ConvStatusPrev1:=fbS2.ConvStatus1,
        ConvStatusPrev2:=fbS2.ConvStatus2, bButtConv:= bButt2s03, bButtConvRev:=bButt2s03Rev, bButtMove:=bButt2s02_s03, 
		 bDirect:=bDirect	,bReverse:=bReverse,
	    bMove1:=bMove2s02_2_s03_1, bMove2:=bMove2s02_s03, bMove3:=bMove2s03_1_s03_2, 
        ConvStatusNext1:= fbS4.ConvStatus1, ConvStatusNext2:= fbS4.ConvStatus2,    
         bEnableMove3:=bEnableMove3_4,  bEnableMove2:= TRUE,  //bSensFreePrev1:=fbS2.bSensFree1, bSensFreePrev2:=fbS2.bSensFree2,
         bLongMove1=> bLongMove2s02_2_s03_1,bLongMove2=>bLongMove2s02_s03, bLongMove3=> bLongMove2s03_1_s03_2   );	  
		
	    bEnableMoveToS4:= NOT bMove2s04_2_s05 AND NOT bMove2s02_2_s03_1 AND NOT bMove2s03_1_s03_2;
		
		
		bEnableMove3_4 := fbS6.ConvStatus=0 OR fbS5.ConvStatus=0 AND NOT (bMove2s05_s06 OR bMove2s04_2_s05);
		
 			
		
		
fbS4 ( bAutomat:=bAutomat, bManual:=bManual,bStop:=bStop,bReset:=bReset, bEnableMove:=bEnableMoveToS4,bBuffering:=bBuffering,
        bDriveMove:=fbS5.bDrivePrev  AND bSens2s05D2, bSens1:=bSens2s04D2, bSens2:=bSens2s04D1,ConvStatusPrev1:=fbS3.ConvStatus1,
        ConvStatusPrev2:=fbS3.ConvStatus2, bButtConv:= bButt2s04, bButtConvRev:=bButt2s04Rev, bButtMove:=bButt2s03_s04, 
		 bDirect:=bDirect	,bReverse:=bReverse,
	    bMove1:=bMove2s03_2_s04_1, bMove2:=bMove2s03_s04, bMove3:=bMove2s04_1_s04_2, 
		ConvStatusNext1:= fbS5.ConvStatus,
          bEnableMove3:=bEnableMove3_4,  bEnableMove2:= TRUE,  //bSensFreePrev1:=fbS3.bSensFree1, bSensFreePrev2:=fbS3.bSensFree2,
         bLongMove1=>bLongMove2s03_2_s04_1,bLongMove2=>bLongMove2s03_s04, bLongMove3=> bLongMove2s04_1_s04_2  );	  
	
  
		
		
		
		bEnableRead := NOT bMove2s05_s06 AND NOT bMove2s03_2_s04_1 AND NOT bMove2s04_1_s04_2 AND NOT bMove2s03_s04;
		
fbLoadScan (bAutomat:=bAutomat,bEnable:=bEnableRead, iConvStatus:=fbS4.ConvStatus2, 
        sInID:=sScanID_2, stLoad:=stLoadS4_2, bReadScan:=bReadScan_2, 
        bRequestID=>bRequestID_2,bEnableReadyID=>bEnableReadyID, bOverflowID=>bOverflow_CTU_ID2,
		bSetVal:=bSetVal_ID2, bResetCTU:=bResetCTU_ID2, bCountNoRead=>bCountNoRead_ID2);		 
		
						
	    bEnableMoveToS5:= NOT bMove2s05_s06 AND NOT bMove2s03_2_s04_1 AND NOT bMove2s04_1_s04_2  AND bEnableReadyID;
	  
fbS5 ( bAutomat:=bAutomat, bManual:=bManual,bStop:=bStop,bReset:=bReset, bEnableMove:= bEnableMoveToS5,
        bDriveMove:=fbS6.bDrivePrev, bSens1:=bSens2s05D2, bSens2:=bSens2s05D1, bStopSecPlace:=TRUE,
        bButtConv:= bButt2s05,bButtConvRev:=bButt2s05Rev, ConvStatusPrev := fbS4.ConvStatus2,
		bSensFreePrev:= bSens2s04D1, bDirect:=bDirect	,bReverse:=bReverse,
	    bMove:=bMove2s04_2_s05, bLongMove=>bLongMove2s04_2_s05, );  
	  	
		
		bEnableWeight := NOT bMove2s04_2_s05 AND NOT bMove2s05_s06 ;
		
fbLoadWeight (bAutomat:=bAutomat,bEnable:=bEnableWeight,bMove:=bMove2s04_2_s05, iConvStatus:=fbS5.ConvStatus, stLoadIn:=stLoadS4_2,
        (*sInWeight:=sWeight_1*)rInWeight:= Massa_2_Gramms   ,  stLoad:=stLoadS5_2, stLoadMove:=stLoadS4_5_2, 
       (* bRequestWeight=>bRequestWeight_1,*) bEnableReadyData=>bEnableReadyData, bOverflowWeight=>bOverflow_CTU_Weight2,
		  bCountNoReadWeight=>bCountNoRead_Weight2, bSetValWeight:=bSetVal_Weight2, bResetCTUWeight:=bResetCTU_Weight2);	
		
			
	    bEnableMoveToS6:= NOT bMove2s04_2_s05   AND bEnableReadyData ;
	  
fbS6 ( bAutomat:=bAutomat, bManual:=bManual,bStop:=bStop,bReset:=bReset, bEnableMove:= bEnableMoveToS6,
        bSens1:=TRUE, bSens2:=bSens2s06D1, bSensFork:= bSens2s06D2, bButtConv:= bButt2s06, bButtConvRev:=bButt2s06Rev,
		 bDirect:=bDirect	,bReverse:=bReverse,  bLastPlace:=TRUE,
	    bMove:=bMove2s05_s06,ConvStatusPrev := fbS5.ConvStatus,bSensFreePrev := bSensFreePrevS6, bLongMove=>bLongMove2s05_1s06,);  
		
		bSensFreePrevS6 := fbS6.ConvStatus = 0;
		
		
fbLoadDataToWMS(bAutomat:=bAutomat,stLoadIn:=stLoadS5_2, bEnable:=NOT bMove2s05_s06, 
iConvStatus:=fbS6.ConvStatus, bMove	:=bMove2s05_s06, stLoadMove:=  stLoadS5_6_2, stLoad:=stLoadS6_2,
sMessageOut=>sMessageOut2, bMessageReady:=bMessageReady2	);			
		
	  
bDrive2s01M1    := fbS1.bDrive 		AND bDirect ;
bDrive2s01M1Rev := fbS1.bDriveRev 		AND bReverse AND bSens2s01D2;
bDrive2s02M1    := fbS2.bDrive 		AND bDirect ;
bDrive2s02M1Rev := fbS2.bDriveReverse 	AND bReverse;
bDrive2s03M1    := fbS3.bDrive 		AND bDirect ;
bDrive2s03M1Rev := fbS3.bDriveReverse 	AND bReverse;
bDrive2s04M1    := fbS4.bDrive 		AND bDirect ;
bDrive2s04M1Rev := fbS4.bDriveReverse 	AND bReverse;  
bDrive2s05M1    := fbS5.bDrive 		AND bDirect ;
bDrive2s05M1Rev := fbS5.bDriveRev 		AND bReverse;
bDrive2s06M1    := fbS6.bDrive 		AND bDirect  AND bSens2s06D1;
bDrive2s06M1Rev := fbS6.bDriveRev 		AND bReverse;

END_PROGRAM

// ---- POUs/ConvLine3.TcPOU
PROGRAM ConvLine3
VAR_INPUT
	bAutomat				:BOOL;
	bManual					:BOOL;
	bStop					:BOOL;
	bReset					:BOOL := FALSE;
	bDirect					:BOOL;
	bReverse				:BOOL;
	bBuffering				:BOOL;
END_VAR
VAR
	fbS1			:FB_ConvPlace;
	fbS2			:FB_ConvPlaceDouble;
	fbS3			:FB_ConvPlaceDouble;
	fbS4			:FB_ConvPlaceDouble;
	fbS5			:FB_ConvPlace;
	fbS6			:FB_ConvPlace;
	bMove1					:BOOL;
	bMove2					:BOOL;
	bDriveMoveS1			:BOOL;
	bDriveMoveS2			:BOOL;
	bEnableMoveToS1			:BOOL :=TRUE;
	bEnableMoveToS2			:BOOL;
	bEnableMoveToS3			:BOOL;
	bEnableMoveToS4			:BOOL;
	bEnableMoveToS5			:BOOL;
	bEnableMoveToS6			:BOOL;
	bEnableRead				:BOOL;
	bEnableWeight			:BOOL;
	fbLoadScan				:FB_LoadScan;
	fbLoadWeight			:FB_LoadWeight;
	bEnableReadyID			:BOOL;
	bEnableReadyData		:BOOL;
	ConvStatusPrev 			:BYTE;
	bSensFreePrevS1 		:BOOL;
	bSensFreePrevS5 		:BOOL;
	bSensFreePrevS6 		:BOOL;

	bCountNoRead_ID1		:WORD;		//Кол-во несчитываний RFID
	bSetVal_ID1				:WORD :=10;	//Заданное значение счетчика (максимально допустимое для несчитываний)
	bResetCTU_ID1			:BOOL;		//Сброс счетчика несчитываний
	
	bCountNoRead_Weight1	:WORD;		//Кол-во несчитываний RFID
	bSetVal_Weight1			:WORD :=10;	//Заданное значение счетчика (максимально допустимое для несчитываний)
	bResetCTU_Weight1		:BOOL;		//Сброс счетчика несчитываний
	
	fbLoadDataToWMS: FB_LoadDataToWMS;
	
	bEnableMove3_2:BOOL;
	bEnableMove3_3:BOOL;
	bEnableMove3_4:BOOL;
	
	fbDelayEnableMove3_2:TON;
	fbDelayEnableMove3_3:TON;
	fbDelayEnableMove3_4:TON;
	
	
	fbFallMove1:F_TRIG;
	fbFallMove2:F_TRIG;
	bLineFree:BOOL;
	fbFreeS6:R_TRIG;
END_VAR
VAR PERSISTENT
	iCounterPallets:INT;
END_VAR




fbS1 ( bAutomat:=bAutomat, bManual:=bManual,bStop:=bStop,bReset:=bReset,tBusy:=T#6S, bFirstPlace:=TRUE,
       	bDriveMove:=fbS2.bDrivePrev, bSens1:=bSens3s01D2, bSens2:=bSens3s01D1, bDirect:=bDirect	,bReverse:=bReverse,
       	bSensFork:= bSens3s01D3, bButtConv:= bButt3s01,bButtConvRev:=bButt3s01Rev,
	  	bMove:=bMove1,ConvStatusPrev:=ConvStatusPrev, bEnableMove := bEnableMoveToS1, bSensFreePrev := bSensFreePrevS1);
	  
		bSensFreePrevS1 := fbS1.ConvStatus = 0;
	  	bEnableMoveToS2:= NOT bMove3s02_2_s03_1 AND NOT bMove3s02_s03;
	  
		bLineFree:= fbS3.ConvStatus1=0 AND fbS3.ConvStatus2=0 AND 
      fbS4.ConvStatus1=0 AND fbS4.ConvStatus2=0 AND NOT (bMove3s02_2_s03_1 OR bMove3s02_s03 OR bMove3s03_1_s03_2
      OR bMove3s03_2_s04_1 OR bMove3s03_s04 OR bMove3s04_1_s04_2  OR bMove3s05_s06 OR bMove3s04_2_s05);	 
	  
 IF bLineFree AND fbS6.ConvStatus=0 AND fbS5.ConvStatus=0 THEN
	 iCounterPallets:=0;
 END_IF
	  
		fbFallMove1(CLK:=bMove3s02_2_s03_1);
IF fbFallMove1.Q THEN	
iCounterPallets:=iCounterPallets +1;
END_IF	
	   fbFallMove2(CLK:=bMove3s02_s03);
IF 	fbFallMove2.Q   THEN
	iCounterPallets:=iCounterPallets +2;
END_IF



		fbFreeS6(CLK:=fbS6.ConvStatus=0);
IF fbFreeS6.Q AND iCounterPallets>0 THEN
iCounterPallets:=iCounterPallets -1;	
END_IF

		
		bEnableMove3_2 := (*(fbS6.ConvStatus=0 OR fbS5.ConvStatus=0) AND bLineFree OR *)iCounterPallets<2;
	//  fbDelayEnableMove3_2(IN:=bEnableMove3_2, PT:=T#0.3S);
		
	  
	
	
	  
fbS2 ( bAutomat:=bAutomat, bManual:=bManual,bStop:=bStop,bReset:=bReset, bEnableMove:=bEnableMoveToS2,bBuffering:=bBuffering,
        bDriveMove:=fbS3.bDrivePrev, bSens1:=bSens3s02D2, bSens2:=bSens3s02D1,bSensFork:= bSens3s01D3, ConvStatusPrev1:=0,
        ConvStatusPrev2:=fbS1.ConvStatus, bButtConv:= bButt3s02, bButtConvRev:=bButt3s02Rev, bButtMove:=bButt3s01_s02,
         bDirect:=bDirect	,bReverse:=bReverse,   ConvStatusNext1:= fbS3.ConvStatus1, ConvStatusNext2:= fbS3.ConvStatus2,
		 bEnableMove3:=bEnableMove3_2(*fbDelayEnableMove3_2.Q*), bEnableMove2:= iCounterPallets>1,  //bSensFreePrev2:=fbS1.bSensFree,
	    bMove1:=bMove3s01_s02_1, bMove2:=bMove2, bMove3:=bMove3s02_1_s02_2, 
        bLongMove1=> bLongMove3s01_s02_1,bLongMove3=> bLongMove3s02_1_s02_2  );

	    bEnableMoveToS3:= NOT bMove3s03_2_s04_1 AND NOT bMove3s03_s04 AND NOT bMove3s01_s02_1 AND NOT bMove3s02_1_s02_2;
 
		
		bEnableMove3_3 := (fbS6.ConvStatus=0 OR fbS5.ConvStatus=0) AND fbS4.ConvStatus1=0 AND fbS4.ConvStatus2=0 
       AND NOT (bMove3s03_2_s04_1 OR bMove3s03_s04 OR bMove3s04_1_s04_2 OR bMove3s05_s06 OR bMove3s04_2_s05);
		  fbDelayEnableMove3_3(IN:=bEnableMove3_3, PT:=T#0.3S);
		  
fbS3 ( bAutomat:=bAutomat, bManual:=bManual,bStop:=bStop,bReset:=bReset, bEnableMove:=bEnableMoveToS3,bBuffering:=bBuffering,
        bDriveMove:=fbS4.bDrivePrev, bSens1:=bSens3s03D2, bSens2:=bSens3s03D1,ConvStatusPrev1:=fbS2.ConvStatus1,
        ConvStatusPrev2:=fbS2.ConvStatus2, bButtConv:= bButt3s03, bButtConvRev:=bButt3s03Rev, bButtMove:=bButt3s02_s03, 
		 bDirect:=bDirect	,bReverse:=bReverse,   ConvStatusNext1:= fbS4.ConvStatus1, ConvStatusNext2:= fbS4.ConvStatus2,
		 bEnableMove3:=fbDelayEnableMove3_3.Q,  bEnableMove2:= TRUE,  //bSensFreePrev1:=fbS2.bSensFree1, bSensFreePrev2:=fbS2.bSensFree2,
	    bMove1:=bMove3s02_2_s03_1, bMove2:=bMove3s02_s03, bMove3:=bMove3s03_1_s03_2, 
        bLongMove1=> bLongMove3s02_2_s03_1,bLongMove2=>bLongMove3s02_s03, bLongMove3=> bLongMove3s03_1_s03_2 );	  
	  
	    bEnableMoveToS4:= NOT bMove3s04_2_s05 AND NOT bMove3s02_2_s03_1 AND NOT bMove3s03_1_s03_2;
 
		
		
		bEnableMove3_4 := fbS6.ConvStatus=0 OR fbS5.ConvStatus=0 AND NOT (bMove3s05_s06 OR bMove3s04_2_s05);
		fbDelayEnableMove3_4(IN:=bEnableMove3_4, PT:=T#0.3S);
		
fbS4 ( bAutomat:=bAutomat, bManual:=bManual,bStop:=bStop,bReset:=bReset, bEnableMove:=bEnableMoveToS4,bBuffering:=bBuffering,
        bDriveMove:=fbS5.bDrivePrev AND bSens3s05D2, bSens1:=bSens3s04D2, bSens2:=bSens3s04D1,ConvStatusPrev1:=fbS3.ConvStatus1,
        ConvStatusPrev2:=fbS3.ConvStatus2, bButtConv:= bButt3s04, bButtConvRev:=bButt3s04Rev, bButtMove:=bButt3s03_s04,
         bDirect:=bDirect	,bReverse:=bReverse,   ConvStatusNext1:= fbS5.ConvStatus,
		 bEnableMove3:=fbDelayEnableMove3_4.Q,  bEnableMove2:= TRUE, // bSensFreePrev1:=fbS3.bSensFree1, bSensFreePrev2:=fbS3.bSensFree2,
	    bMove1:=bMove3s03_2_s04_1, bMove2:=bMove3s03_s04, bMove3:=bMove3s04_1_s04_2, 
         bLongMove1=>bLongMove3s03_2_s04_1,bLongMove2=>bLongMove3s03_s04, bLongMove3=> bLongMove3s04_1_s04_2  );	  
	
  		
		bEnableRead := NOT bMove3s05_s06 AND NOT bMove3s03_2_s04_1 AND NOT bMove3s04_1_s04_2 AND NOT bMove3s03_s04 ;
		
fbLoadScan (bAutomat:=bAutomat,bEnable:=bEnableRead, iConvStatus:=fbS4.ConvStatus2, 
        sInID:=sScanID_1, stLoad:=stLoadS4_1, bReadScan:=bReadScan_1, 
        bRequestID=>bRequestID_1,bEnableReadyID=>bEnableReadyID, bOverflowID=>bOverflow_CTU_ID1,
		bSetVal:=bSetVal_ID1, bResetCTU:=bResetCTU_ID1, bCountNoRead=>bCountNoRead_ID1);		 
		
						
	    bEnableMoveToS5:= NOT bMove3s05_s06 AND NOT bMove3s03_2_s04_1 AND NOT bMove3s04_1_s04_2  AND bEnableReadyID;
	  
fbS5 ( bAutomat:=bAutomat, bManual:=bManual,bStop:=bStop,bReset:=bReset, bEnableMove:= bEnableMoveToS5,
        bDriveMove:=fbS6.bDrivePrev, bSens1:=bSens3s05D2, bSens2:=bSens3s05D1, bStopSecPlace:=TRUE,
        bButtConv:= bButt3s05,bButtConvRev:=bButt3s05Rev, ConvStatusPrev := fbS4.ConvStatus2,
		 bDirect:=bDirect	,bReverse:=bReverse,
		bSensFreePrev:= bSens3s04D1, bMove:=bMove3s04_2_s05,bLongMove=>bLongMove3s04_2_s05, );  
	  	
	
		bEnableWeight := NOT bMove3s04_2_s05 AND NOT bMove3s05_s06 ;
		
fbLoadWeight (bAutomat:=bAutomat,bEnable:=bEnableWeight,bMove:=bMove3s04_2_s05, iConvStatus:=fbS5.ConvStatus, stLoadIn:=stLoadS4_1,
        (*sInWeight:=sWeight_1*)rInWeight:= Massa_1_Gramms   ,  stLoad:=stLoadS5_1, stLoadMove:=stLoadS4_5_1, 
        (*bRequestWeight=>bRequestWeight_1,*) bEnableReadyData=>bEnableReadyData, bOverflowWeight=>bOverflow_CTU_Weight1,
		  bCountNoReadWeight=>bCountNoRead_Weight1, bSetValWeight:=bSetVal_Weight1, bResetCTUWeight:=bResetCTU_Weight1);	
		
			
	    bEnableMoveToS6:= NOT bMove3s04_2_s05   AND bEnableReadyData ;
	  
fbS6 ( bAutomat:=bAutomat, bManual:=bManual,bStop:=bStop,bReset:=bReset, bEnableMove:= bEnableMoveToS6,
        bSens1:=TRUE, bSens2:=bSens3s06D1, (*bSensFork:= bSens3s06D2, *)bButtConv:= bButt3s06, bButtConvRev:=bButt3s06Rev,
		 bDirect:=bDirect	,bReverse:=bReverse,bLastPlace:=TRUE,bLongMove=>bLongMove3s05_1s06,
	    bMove:=bMove3s05_s06,ConvStatusPrev := fbS5.ConvStatus,bSensFreePrev := bSensFreePrevS6);  
		
		bSensFreePrevS6 := fbS6.ConvStatus = 0;
		
		
fbLoadDataToWMS(bAutomat:=bAutomat,stLoadIn:=stLoadS5_1, bEnable:=NOT bMove3s05_s06, 
iConvStatus:=fbS6.ConvStatus, bMove	:=bMove3s05_s06, stLoadMove:=  stLoadS5_6_1, stLoad:=stLoadS6_1,
sMessageOut=>sMessageOut1, bMessageReady:=bMessageReady1	);		
		
		
	  
bDrive3s01M1    := fbS1.bDrive 		AND bDirect ;
bDrive3s01M1Rev := fbS1.bDriveRev 		AND bReverse AND bSens3s01D2;
bDrive3s02M1    := fbS2.bDrive 		AND bDirect ;
bDrive3s02M1Rev := fbS2.bDriveReverse 	AND bReverse;
bDrive3s03M1    := fbS3.bDrive 		AND bDirect ;
bDrive3s03M1Rev := fbS3.bDriveReverse 	AND bReverse;
bDrive3s04M1    := fbS4.bDrive 		AND bDirect ;
bDrive3s04M1Rev := fbS4.bDriveReverse 	AND bReverse;  
bDrive3s05M1    := fbS5.bDrive 		AND bDirect ;
bDrive3s05M1Rev := fbS5.bDriveRev 		AND bReverse;
bDrive3s06M1    := fbS6.bDrive 		AND bDirect AND bSens3s06D1;
bDrive3s06M1Rev := fbS6.bDriveRev 		AND bReverse;

END_PROGRAM

// ---- POUs/ConvLine4.TcPOU
PROGRAM ConvLine4
VAR_INPUT
	bAutomat				:BOOL;
	bManual					:BOOL;
	bStop					:BOOL;
	bReset					:BOOL := FALSE;
	bDirect					:BOOL;
	bReverse				:BOOL;
	bBuffering				:BOOL;
END_VAR
VAR
	fbS1			:FB_ConvPlace;
	fbS2			:FB_ConvPlaceDouble;
	fbS3			:FB_ConvPlaceDouble;
	fbS4			:FB_ConvPlaceDouble;
	fbS5			:FB_ConvPlace;
	fbS6			:FB_ConvPlace;
	bMove1					:BOOL;
	bMove2					:BOOL;
	bDriveMoveS1			:BOOL;
	bDriveMoveS2			:BOOL;
	bEnableMoveToS1			:BOOL :=TRUE;
	bEnableMoveToS2			:BOOL;
	bEnableMoveToS3			:BOOL;
	bEnableMoveToS4			:BOOL;
	bEnableMoveToS5			:BOOL;
	bEnableMoveToS6			:BOOL;
	bEnableRead				:BOOL;
	bEnableWeight			:BOOL;
	fbLoadScan				:FB_LoadScan;
	fbLoadWeight			:FB_LoadWeight;
	bEnableReadyID			:BOOL;
	bEnableReadyData		:BOOL;
	ConvStatusPrev 			:BYTE;
	bSensFreePrevS1 		:BOOL;
	bSensFreePrevS5 		:BOOL;
	bSensFreePrevS6 		:BOOL;

	bCountNoRead_ID1		:WORD;		//Кол-во несчитываний RFID
	bSetVal_ID1				:WORD :=10;	//Заданное значение счетчика (максимально допустимое для несчитываний)
	bResetCTU_ID1			:BOOL;		//Сброс счетчика несчитываний
	
	bCountNoRead_Weight1	:WORD;		//Кол-во несчитываний RFID
	bSetVal_Weight1			:WORD :=10;	//Заданное значение счетчика (максимально допустимое для несчитываний)
	bResetCTU_Weight1		:BOOL;		//Сброс счетчика несчитываний
	
	fbLoadDataToWMS: FB_LoadDataToWMS;
	
	bEnableMove3_2:BOOL;
	bEnableMove3_3:BOOL;
	bEnableMove3_4:BOOL;
	
	fbDelayEnableMove3_2:TON;
	fbDelayEnableMove3_3:TON;
	fbDelayEnableMove3_4:TON;
	
	
	fbFallMove1:F_TRIG;
	fbFallMove2:F_TRIG;
	bLineFree:BOOL;
	fbFreeS6:R_TRIG;
END_VAR
VAR PERSISTENT
	iCounterPallets:INT;
END_VAR




fbS1 ( bAutomat:=bAutomat, bManual:=bManual,bStop:=bStop,bReset:=bReset,tBusy:=T#6S, bFirstPlace:=TRUE,
       	bDriveMove:=fbS2.bDrivePrev, bSens1:=bSens4s01D2, bSens2:=bSens4s01D1, bDirect:=bDirect	,bReverse:=bReverse,
       	bSensFork:= bSens4s01D3, bButtConv:= bButt4s01,bButtConvRev:=bButt4s01Rev,
	  	bMove:=bMove1,ConvStatusPrev:=ConvStatusPrev, bEnableMove := bEnableMoveToS1, bSensFreePrev := bSensFreePrevS1);
	  
		bSensFreePrevS1 := fbS1.ConvStatus = 0;
	  	bEnableMoveToS2:= NOT bMove4s02_2_s03_1 AND NOT bMove4s02_s03;
	  
		bLineFree:= fbS3.ConvStatus1=0 AND fbS3.ConvStatus2=0 AND 
      fbS4.ConvStatus1=0 AND fbS4.ConvStatus2=0 AND NOT (bMove4s02_2_s03_1 OR bMove4s02_s03 OR bMove4s03_1_s03_2
      OR bMove4s03_2_s04_1 OR bMove4s03_s04 OR bMove4s04_1_s04_2  OR bMove4s05_s06 OR bMove4s04_2_s05);	 
	  
 IF bLineFree AND fbS6.ConvStatus=0 AND fbS5.ConvStatus=0 THEN
	 iCounterPallets:=0;
 END_IF
	  
		fbFallMove1(CLK:=bMove4s02_2_s03_1);
IF fbFallMove1.Q THEN	
iCounterPallets:=iCounterPallets +1;
END_IF	
	   fbFallMove2(CLK:=bMove4s02_s03);
IF 	fbFallMove2.Q   THEN
	iCounterPallets:=iCounterPallets +2;
END_IF



		fbFreeS6(CLK:=fbS6.ConvStatus=0);
IF fbFreeS6.Q AND iCounterPallets>0 THEN
iCounterPallets:=iCounterPallets -1;	
END_IF

		
		bEnableMove3_2 := (*(fbS6.ConvStatus=0 OR fbS5.ConvStatus=0) AND bLineFree OR *)iCounterPallets<2;
	//  fbDelayEnableMove3_2(IN:=bEnableMove3_2, PT:=T#0.3S);
		
	  
	
	
	  
fbS2 ( bAutomat:=bAutomat, bManual:=bManual,bStop:=bStop,bReset:=bReset, bEnableMove:=bEnableMoveToS2,bBuffering:=bBuffering,
        bDriveMove:=fbS3.bDrivePrev, bSens1:=bSens4s02D2, bSens2:=bSens4s02D1,bSensFork:= bSens4s01D3, ConvStatusPrev1:=0,
        ConvStatusPrev2:=fbS1.ConvStatus, bButtConv:= bButt4s02, bButtConvRev:=bButt4s02Rev, bButtMove:=bButt4s01_s02,
         bDirect:=bDirect	,bReverse:=bReverse,   ConvStatusNext1:= fbS3.ConvStatus1, ConvStatusNext2:= fbS3.ConvStatus2,
		 bEnableMove3:=bEnableMove3_2(*fbDelayEnableMove3_2.Q*), bEnableMove2:= iCounterPallets>1,  //bSensFreePrev2:=fbS1.bSensFree,
	    bMove1:=bMove4s01_s02_1, bMove2:=bMove2, bMove3:=bMove4s02_1_s02_2, 
        bLongMove1=> bLongMove4s01_s02_1,bLongMove3=> bLongMove4s02_1_s02_2  );

	    bEnableMoveToS3:= NOT bMove4s03_2_s04_1 AND NOT bMove4s03_s04 AND NOT bMove4s01_s02_1 AND NOT bMove4s02_1_s02_2;
 
		
		bEnableMove3_3 := (fbS6.ConvStatus=0 OR fbS5.ConvStatus=0) AND fbS4.ConvStatus1=0 AND fbS4.ConvStatus2=0 
       AND NOT (bMove4s03_2_s04_1 OR bMove4s03_s04 OR bMove4s04_1_s04_2 OR bMove4s05_s06 OR bMove4s04_2_s05);
		  fbDelayEnableMove3_3(IN:=bEnableMove3_3, PT:=T#0.3S);
		  
fbS3 ( bAutomat:=bAutomat, bManual:=bManual,bStop:=bStop,bReset:=bReset, bEnableMove:=bEnableMoveToS3,bBuffering:=bBuffering,
        bDriveMove:=fbS4.bDrivePrev, bSens1:=bSens4s03D2, bSens2:=bSens4s03D1,ConvStatusPrev1:=fbS2.ConvStatus1,
        ConvStatusPrev2:=fbS2.ConvStatus2, bButtConv:= bButt4s03, bButtConvRev:=bButt4s03Rev, bButtMove:=bButt4s02_s03, 
		 bDirect:=bDirect	,bReverse:=bReverse,   ConvStatusNext1:= fbS4.ConvStatus1, ConvStatusNext2:= fbS4.ConvStatus2,
		 bEnableMove3:=fbDelayEnableMove3_3.Q,  bEnableMove2:= TRUE,  //bSensFreePrev1:=fbS2.bSensFree1, bSensFreePrev2:=fbS2.bSensFree2,
	    bMove1:=bMove4s02_2_s03_1, bMove2:=bMove4s02_s03, bMove3:=bMove4s03_1_s03_2, 
        bLongMove1=> bLongMove4s02_2_s03_1,bLongMove2=>bLongMove4s02_s03, bLongMove3=> bLongMove4s03_1_s03_2 );	  
	  
	    bEnableMoveToS4:= NOT bMove4s04_2_s05 AND NOT bMove4s02_2_s03_1 AND NOT bMove4s03_1_s03_2;
 
		
		
		bEnableMove3_4 := fbS6.ConvStatus=0 OR fbS5.ConvStatus=0 AND NOT (bMove4s05_s06 OR bMove4s04_2_s05);
		fbDelayEnableMove3_4(IN:=bEnableMove3_4, PT:=T#0.3S);
		
fbS4 ( bAutomat:=bAutomat, bManual:=bManual,bStop:=bStop,bReset:=bReset, bEnableMove:=bEnableMoveToS4,bBuffering:=bBuffering,
        bDriveMove:=fbS5.bDrivePrev AND bSens4s05D2, bSens1:=bSens4s04D2, bSens2:=bSens4s04D1,ConvStatusPrev1:=fbS3.ConvStatus1,
        ConvStatusPrev2:=fbS3.ConvStatus2, bButtConv:= bButt4s04, bButtConvRev:=bButt4s04Rev, bButtMove:=bButt4s03_s04,
         bDirect:=bDirect	,bReverse:=bReverse,   ConvStatusNext1:= fbS5.ConvStatus,
		 bEnableMove3:=fbDelayEnableMove3_4.Q,  bEnableMove2:= TRUE, // bSensFreePrev1:=fbS3.bSensFree1, bSensFreePrev2:=fbS3.bSensFree2,
	    bMove1:=bMove4s03_2_s04_1, bMove2:=bMove4s03_s04, bMove3:=bMove4s04_1_s04_2, 
         bLongMove1=>bLongMove4s03_2_s04_1,bLongMove2=>bLongMove4s03_s04, bLongMove3=> bLongMove4s04_1_s04_2  );	  
	
  		
		bEnableRead := NOT bMove4s05_s06 AND NOT bMove4s03_2_s04_1 AND NOT bMove4s04_1_s04_2 AND NOT bMove4s03_s04 ;
		
fbLoadScan (bAutomat:=bAutomat,bEnable:=bEnableRead, iConvStatus:=fbS4.ConvStatus2, 
        sInID:=sScanID_1, stLoad:=stLoadS4_1, bReadScan:=bReadScan_1, 
        bRequestID=>bRequestID_1,bEnableReadyID=>bEnableReadyID, bOverflowID=>bOverflow_CTU_ID1,
		bSetVal:=bSetVal_ID1, bResetCTU:=bResetCTU_ID1, bCountNoRead=>bCountNoRead_ID1);		 
		
						
	    bEnableMoveToS5:= NOT bMove4s05_s06 AND NOT bMove4s03_2_s04_1 AND NOT bMove4s04_1_s04_2  AND bEnableReadyID;
	  
fbS5 ( bAutomat:=bAutomat, bManual:=bManual,bStop:=bStop,bReset:=bReset, bEnableMove:= bEnableMoveToS5,
        bDriveMove:=fbS6.bDrivePrev, bSens1:=bSens4s05D2, bSens2:=bSens4s05D1, bStopSecPlace:=TRUE,
        bButtConv:= bButt4s05,bButtConvRev:=bButt4s05Rev, ConvStatusPrev := fbS4.ConvStatus2,
		 bDirect:=bDirect	,bReverse:=bReverse,
		bSensFreePrev:= bSens4s04D1, bMove:=bMove4s04_2_s05,bLongMove=>bLongMove4s04_2_s05, );  
	  	
	
		bEnableWeight := NOT bMove4s04_2_s05 AND NOT bMove4s05_s06 ;
		
fbLoadWeight (bAutomat:=bAutomat,bEnable:=bEnableWeight,bMove:=bMove4s04_2_s05, iConvStatus:=fbS5.ConvStatus, stLoadIn:=stLoadS4_1,
        (*sInWeight:=sWeight_1*)rInWeight:= Massa_1_Gramms   ,  stLoad:=stLoadS5_1, stLoadMove:=stLoadS4_5_1, 
        (*bRequestWeight=>bRequestWeight_1,*) bEnableReadyData=>bEnableReadyData, bOverflowWeight=>bOverflow_CTU_Weight1,
		  bCountNoReadWeight=>bCountNoRead_Weight1, bSetValWeight:=bSetVal_Weight1, bResetCTUWeight:=bResetCTU_Weight1);	
		
			
	    bEnableMoveToS6:= NOT bMove4s04_2_s05   AND bEnableReadyData ;
	  
fbS6 ( bAutomat:=bAutomat, bManual:=bManual,bStop:=bStop,bReset:=bReset, bEnableMove:= bEnableMoveToS6,
        bSens1:=TRUE, bSens2:=bSens4s06D1, (*bSensFork:= bSens4s06D2, *)bButtConv:= bButt4s06, bButtConvRev:=bButt4s06Rev,
		 bDirect:=bDirect	,bReverse:=bReverse,bLastPlace:=TRUE,bLongMove=>bLongMove4s05_1s06,
	    bMove:=bMove4s05_s06,ConvStatusPrev := fbS5.ConvStatus,bSensFreePrev := bSensFreePrevS6);  
		
		bSensFreePrevS6 := fbS6.ConvStatus = 0;
		
		
fbLoadDataToWMS(bAutomat:=bAutomat,stLoadIn:=stLoadS5_1, bEnable:=NOT bMove4s05_s06, 
iConvStatus:=fbS6.ConvStatus, bMove	:=bMove4s05_s06, stLoadMove:=  stLoadS5_6_1, stLoad:=stLoadS6_1,
sMessageOut=>sMessageOut1, bMessageReady:=bMessageReady1	);		
		
		
	  
bDrive4s01M1    := fbS1.bDrive 		AND bDirect ;
bDrive4s01M1Rev := fbS1.bDriveRev 		AND bReverse AND bSens4s01D2;
bDrive4s02M1    := fbS2.bDrive 		AND bDirect ;
bDrive4s02M1Rev := fbS2.bDriveReverse 	AND bReverse;
bDrive4s03M1    := fbS3.bDrive 		AND bDirect ;
bDrive4s03M1Rev := fbS3.bDriveReverse 	AND bReverse;
bDrive4s04M1    := fbS4.bDrive 		AND bDirect ;
bDrive4s04M1Rev := fbS4.bDriveReverse 	AND bReverse;  
bDrive4s05M1    := fbS5.bDrive 		AND bDirect ;
bDrive4s05M1Rev := fbS5.bDriveRev 		AND bReverse;
bDrive4s06M1    := fbS6.bDrive 		AND bDirect AND bSens4s06D1;
bDrive4s06M1Rev := fbS6.bDriveRev 		AND bReverse;

END_PROGRAM
